// TIA Portal V17 export
// export: Created 2023-12-22T15:28:35.5105412Z, ExportSetting WithDefaults, DisplayName Totally Integrated Automation Portal, DisplayVersion V17, DisplayName TIA Portal Openness, DisplayVersion V17, DisplayName TIA Portal Version Control Interface, DisplayVersion V17, DisplayName STEP 7 Professional, DisplayVersion V17, DisplayName STEP 7 Safety, DisplayVersion V17, DisplayName WinCC Advanced, DisplayVersion V17
FUNCTION_BLOCK "AIx"   // FB220, LAD
{ S7_Optimized_Access := 'FALSE' }
VERSION : 0.1
// Signal - PIW код сигнала от датчика
// pulse - частота алгоритма фильтрации
// Result - результат обработки сигнала, формат Real
// stored: AutoNumber false, IsIECCheckEnabled false, SetENOAutomatically false, UDAEnableTagReadback false
   VAR DB_SPECIFIC
      Time_DTL { S7_SetPoint := 'True'} : DTL;
   END_VAR
BEGIN

REGION Network 1: Датчик уровня
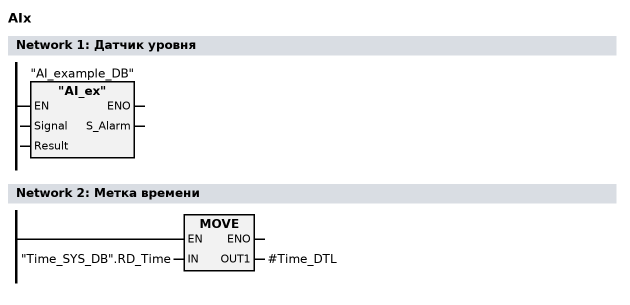
   RUNG wire#powerrail
      "AI_example_DB"(Signal :=, Result :=, S_Alarm =>)
   END_RUNG
   // the same network as SCL:
   "AI_example_DB"();   // "AI_ex"
END_REGION

REGION Network 2: Метка времени
   RUNG wire#powerrail
      Move(in := "Time_SYS_DB".RD_Time, out1 => #Time_DTL)
   END_RUNG
   // the same network as SCL:
   #Time_DTL := "Time_SYS_DB".RD_Time;
END_REGION
END_FUNCTION_BLOCK
